// TIA Portal project "7_Height_Sorting_Basic" (V19)

(* hardware
DEVICE "S7-1500/ET200MP station_1"  S7-1500 station
   slot 0: "Rail_0"  Rack  6ES7 590-1***0-0AA0
   slot 1: "PLC_1"  CPU 1513-1 PN  6ES7 513-1AL02-0AB0  V2.9
      slot 3: "CPU display_1"  6ES7591-1AA00-0AA0
      slot 32768: "PROFINET interface_1"  X1
         slot 32769: "Port_1"  X1 P1
         slot 32770: "Port_2"  X1 P2
      slot 34817: "Virtual CP interface port_1"  Virtual CP interface port  Virtual CP interface port
*)

// ===== PLC "PLC_1"  CPU 1513-1 PN =====

VAR_GLOBAL   // PLC tag table "Default tag table"
   "Tag_1" AT %M0.0 : Bool;
   "Tag_2" AT %M0.1 : Bool;
   "Tag_3" AT %M0.2 : Bool;
   "Tag_4" AT %M0.3 : Bool;
   "Tag_5" AT %M0.4 : Bool;
   "Tag_6" AT %M0.5 : Bool;
   "Tag_7" AT %M2.1 : Bool;
   "Tag_8" AT %M1.7 : Bool;
   "Tag_9" AT %M2.0 : Bool;
   "Tag_10" AT %MW100 : Int;
   "Tag_11" AT %M2.2 : Bool;
   "Tag_12" AT %M1.0 : Bool;
   "Tag_13" AT %M1.1 : Bool;
   "Tag_14" AT %M1.4 : Bool;
   "Tag_15" AT %M1.2 : Bool;
   "Tag_16" AT %M1.3 : Bool;
   "Tag_17" AT %M1.5 : Bool;
   "Tag_18" AT %M1.6 : Bool;
   "Tag_19" AT %M2.4 : Bool;
   "Tag_20" AT %M2.5 : Bool;
END_VAR

VAR_GLOBAL   // PLC tag table "Tag table from XML_1"
   "Start Button" AT %I0.0 : Bool;
   "Stop Button" AT %I0.1 : Bool;
   "High Sensor" AT %I0.2 : Bool;
   "Low Sensor" AT %I0.3 : Bool;
   "Pallet sensor" AT %I0.4 : Bool;
   "Loaded" AT %I0.5 : Bool;
   "At right entry" AT %I0.6 : Bool;
   "At left entry" AT %I0.7 : Bool;
   "At right exit" AT %I1.0 : Bool;
   "At left exit" AT %I1.1 : Bool;
   "Start Button (LED)" AT %Q0.0 : Bool;
   "Stop Button (LED)" AT %Q0.1 : Bool;
   "Conveyor entry" AT %Q0.2 : Bool;
   "Conveyor right" AT %Q0.3 : Bool;
   "Conveyor left" AT %Q0.4 : Bool;
   "Load" AT %Q0.5 : Bool;
   "Transf. left" AT %Q0.6 : Bool;
   "Transf. right" AT %Q0.7 : Bool;
   "Right count" AT %QW30 : Int;
   "Left Count" AT %QW32 : Int;
END_VAR

// folder: System blocks/Program resources

DATA_BLOCK "IEC_Timer_0_DB"   // DB1
{ S7_Optimized_Access := 'TRUE' }
AUTHOR : Simatic
FAMILY : IEC
NAME : IEC_TMR
VERSION : 1.0
// stored: InstanceOfName IEC_TIMER
"IEC_TIMER"
BEGIN
END_DATA_BLOCK

DATA_BLOCK "IEC_Counter_0_DB"   // DB2
{ S7_Optimized_Access := 'TRUE' }
AUTHOR : Simatic
FAMILY : IEC
NAME : CNTR
VERSION : 1.0
// stored: InstanceOfName IEC_COUNTER
"IEC_COUNTER"
BEGIN
END_DATA_BLOCK

DATA_BLOCK "IEC_Counter_0_DB_1"   // DB3
{ S7_Optimized_Access := 'TRUE' }
AUTHOR : Simatic
FAMILY : IEC
NAME : CNTR
VERSION : 1.0
// stored: InstanceOfName IEC_COUNTER
"IEC_COUNTER"
BEGIN
END_DATA_BLOCK

DATA_BLOCK "IEC_Counter_0_DB_2"   // DB4
{ S7_Optimized_Access := 'TRUE' }
AUTHOR : Simatic
FAMILY : IEC
NAME : CNTR
VERSION : 1.0
// stored: InstanceOfName IEC_COUNTER
"IEC_COUNTER"
BEGIN
END_DATA_BLOCK

DATA_BLOCK "IEC_Counter_0_DB_3"   // DB5
{ S7_Optimized_Access := 'TRUE' }
AUTHOR : Simatic
FAMILY : IEC
NAME : CNTR
VERSION : 1.0
// stored: InstanceOfName IEC_COUNTER
"IEC_COUNTER"
BEGIN
END_DATA_BLOCK

// folder: (top level)

ORGANIZATION_BLOCK "Main"   // OB1, LAD, ProgramCycle
TITLE = "Main Program Sweep (Cycle)"
{ S7_Optimized_Access := 'TRUE' }
VERSION : 0.1
   VAR_INPUT
      Initial_Call : Bool;   // Initial call of this OB
      Remanence : Bool;   // =True, if remanent data are available
   END_VAR
   VAR_TEMP   // added for the SCL form of the ladder/FBD networks
      _w1 : Bool;
      _w2 : Bool;
      _w3 : Bool;
      _w4 : Bool;
   END_VAR
BEGIN

REGION Network 1: ON/OFF the LEDs
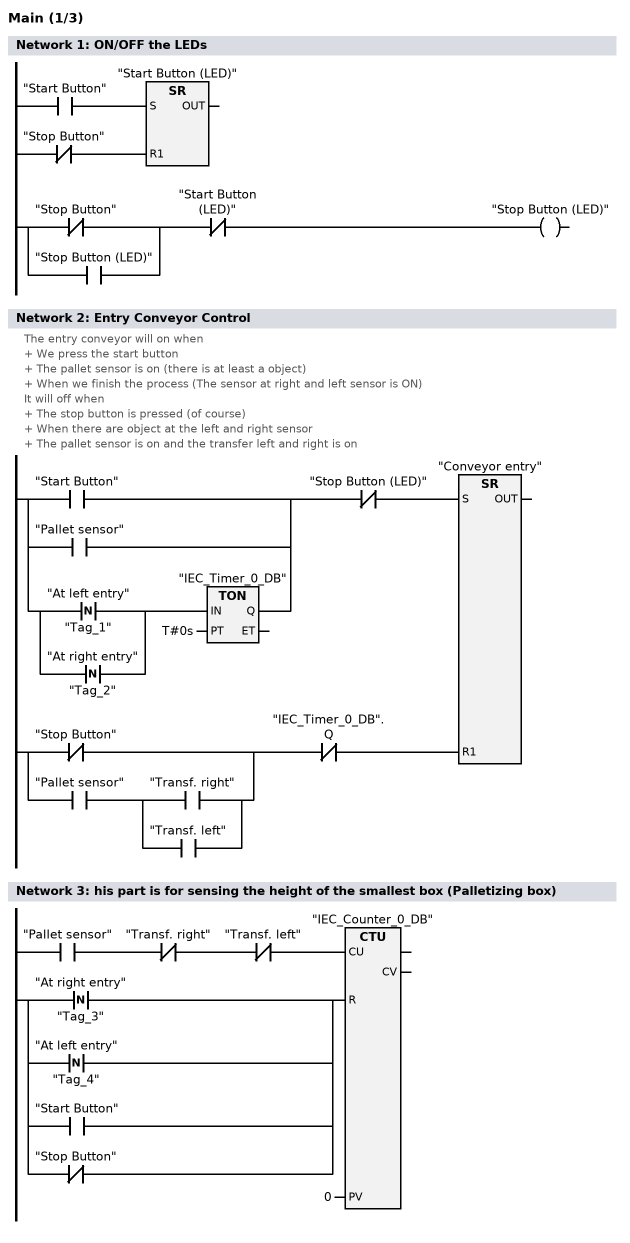
   RUNG wire#powerrail
      Contact( "Start Button" )
      S_SR(operand := "Start Button (LED)", r1 := wire#w1)
   END_RUNG
   RUNG wire#powerrail
      I_Contact( "Stop Button" )
   END_RUNG wire#w1
   RUNG wire#powerrail
      I_Contact( "Stop Button" )
      wire#w2
      I_Contact( "Start Button (LED)" )
      Coil( "Stop Button (LED)" )
   END_RUNG
   RUNG wire#powerrail
      Contact( "Stop Button (LED)" )
   END_RUNG wire#w2
   // the same network as SCL:
   IF "Start Button" THEN
       "Start Button (LED)" := TRUE;   // SR flip-flop
   END_IF;
   IF NOT "Stop Button" THEN "Start Button (LED)" := FALSE; END_IF;
   "Stop Button (LED)" := (NOT "Stop Button" OR "Stop Button (LED)") AND NOT "Start Button (LED)";
END_REGION

REGION Network 2: Entry Conveyor Control
   // The entry conveyor will on when
   // + We press the start button
   // + The pallet sensor is on (there is at least a object)
   // + When we finish the process (The sensor at right and left sensor is ON)
   // It will off when
   // + The stop button is pressed (of course)
   // + When there are object at the left and right sensor
   // + The pallet sensor is on and the transfer left and right is on
   #_w1 := NOT "At left entry" AND "Tag_1";   // falling edge of "At left entry"
   "Tag_1" := "At left entry";
   #_w2 := NOT "At right entry" AND "Tag_2";   // falling edge of "At right entry"
   "Tag_2" := "At right entry";
   "IEC_Timer_0_DB".TON(IN := #_w1 OR #_w2, PT := T#0s);
   IF ("Start Button" OR "Pallet sensor" OR "IEC_Timer_0_DB".Q) AND NOT "Stop Button (LED)" THEN
       "Conveyor entry" := TRUE;   // SR flip-flop
   END_IF;
   IF (NOT "Stop Button" OR ("Pallet sensor" AND ("Transf. right" OR "Transf. left"))) AND NOT "IEC_Timer_0_DB".Q THEN
       "Conveyor entry" := FALSE;
   END_IF;
END_REGION

REGION Network 3: his part is for sensing the height of the smallest box (Palletizing box)
   #_w1 := NOT "At right entry" AND "Tag_3";   // falling edge of "At right entry"
   "Tag_3" := "At right entry";
   #_w2 := NOT "At left entry" AND "Tag_4";   // falling edge of "At left entry"
   "Tag_4" := "At left entry";
   "IEC_Counter_0_DB".CTU(CU := "Pallet sensor" AND NOT "Transf. right" AND NOT "Transf. left",
                          R := #_w1 OR #_w2 OR "Start Button" OR NOT "Stop Button",
                          PV := 0);
END_REGION

REGION Network 4: This part for box size S and M
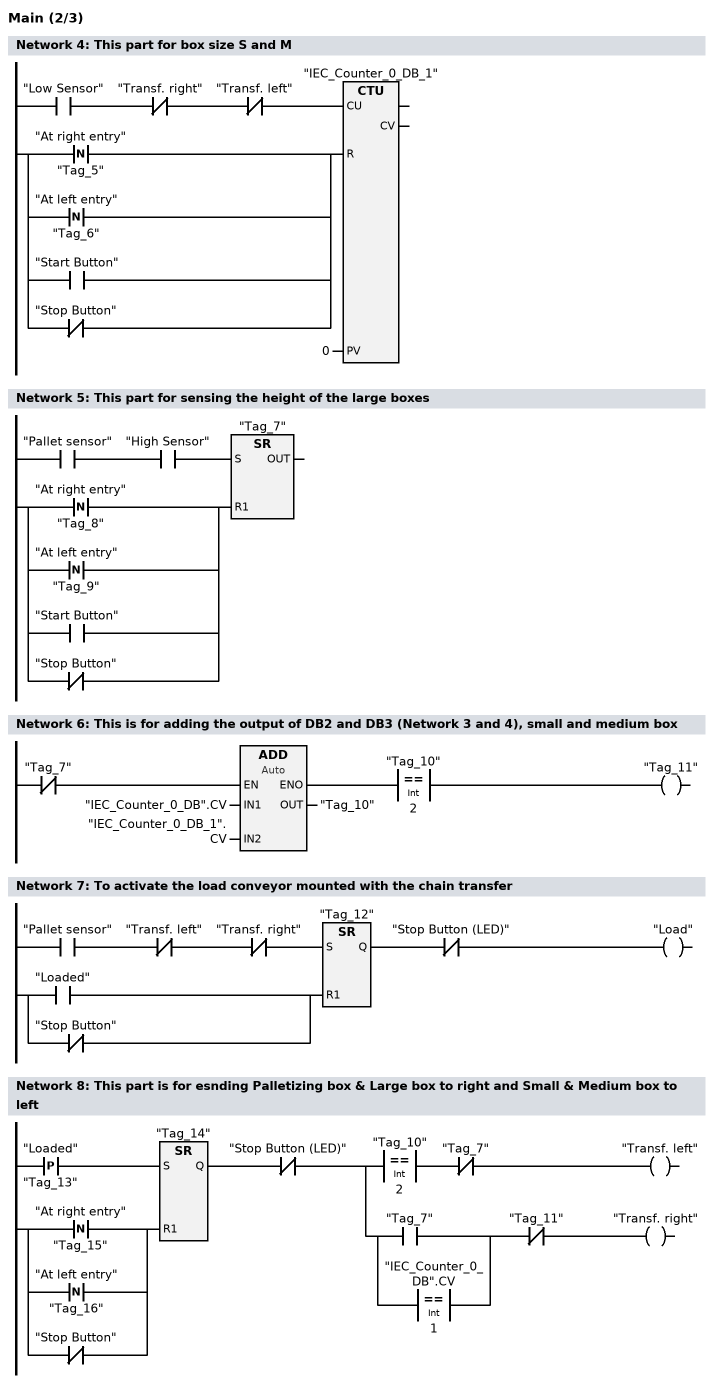
   #_w1 := NOT "At right entry" AND "Tag_5";   // falling edge of "At right entry"
   "Tag_5" := "At right entry";
   #_w2 := NOT "At left entry" AND "Tag_6";   // falling edge of "At left entry"
   "Tag_6" := "At left entry";
   "IEC_Counter_0_DB_1".CTU(CU := "Low Sensor" AND NOT "Transf. right" AND NOT "Transf. left",
                           R := #_w1 OR #_w2 OR "Start Button" OR NOT "Stop Button",
                           PV := 0);
END_REGION

REGION Network 5: This part for sensing the height of the large boxes
   RUNG wire#powerrail
      Contact( "Pallet sensor" )
      Contact( "High Sensor" )
      S_SR(operand := "Tag_7", r1 := wire#w1)
   END_RUNG
   RUNG wire#powerrail
      N_Contact(operand := "At right entry", bit := "Tag_8")
   END_RUNG wire#w1
   RUNG wire#powerrail
      N_Contact(operand := "At left entry", bit := "Tag_9")
   END_RUNG wire#w1
   RUNG wire#powerrail
      Contact( "Start Button" )
   END_RUNG wire#w1
   RUNG wire#powerrail
      I_Contact( "Stop Button" )
   END_RUNG wire#w1
   // the same network as SCL:
   #_w1 := NOT "At right entry" AND "Tag_8";   // falling edge of "At right entry"
   "Tag_8" := "At right entry";
   #_w2 := NOT "At left entry" AND "Tag_9";   // falling edge of "At left entry"
   "Tag_9" := "At left entry";
   IF "Pallet sensor" AND "High Sensor" THEN
       "Tag_7" := TRUE;   // SR flip-flop
   END_IF;
   IF #_w1 OR #_w2 OR "Start Button" OR NOT "Stop Button" THEN "Tag_7" := FALSE; END_IF;
END_REGION

REGION Network 6: This is for adding the output of DB2 and DB3 (Network 3 and 4), small and medium box
   RUNG wire#powerrail
      I_Contact( "Tag_7" )
      Add(in1 := "IEC_Counter_0_DB".CV, in2 := "IEC_Counter_0_DB_1".CV, out => "Tag_10")
      { S7_Templates := "SrcType := Int" } EQ_Contact(in1 := "Tag_10", in2 := 2)
      Coil( "Tag_11" )
   END_RUNG
   // the same network as SCL:
   IF NOT "Tag_7" THEN "Tag_10" := "IEC_Counter_0_DB".CV + "IEC_Counter_0_DB_1".CV; END_IF;
   "Tag_11" := NOT "Tag_7" AND ("Tag_10" = 2);
END_REGION

REGION Network 7: To activate the load conveyor mounted with the chain transfer
   RUNG wire#powerrail
      Contact( "Pallet sensor" )
      I_Contact( "Transf. left" )
      I_Contact( "Transf. right" )
      S_SR(operand := "Tag_12", r1 := wire#w1)
      I_Contact( "Stop Button (LED)" )
      Coil( "Load" )
   END_RUNG
   RUNG wire#powerrail
      Contact( "Loaded" )
   END_RUNG wire#w1
   RUNG wire#powerrail
      I_Contact( "Stop Button" )
   END_RUNG wire#w1
   // the same network as SCL:
   IF "Pallet sensor" AND NOT "Transf. left" AND NOT "Transf. right" THEN
       "Tag_12" := TRUE;   // SR flip-flop
   END_IF;
   IF "Loaded" OR NOT "Stop Button" THEN "Tag_12" := FALSE; END_IF;
   "Load" := "Tag_12" AND NOT "Stop Button (LED)";
END_REGION

REGION Network 8: This part is for esnding Palletizing box & Large box to right and Small & Medium box to left
   RUNG wire#powerrail
      P_Contact(operand := "Loaded", bit := "Tag_13")
      S_SR(operand := "Tag_14", r1 := wire#w1)
      I_Contact( "Stop Button (LED)" )
      wire#w2
      { S7_Templates := "SrcType := Int" } EQ_Contact(in1 := "Tag_10", in2 := 2)
      I_Contact( "Tag_7" )
      Coil( "Transf. left" )
   END_RUNG
   RUNG wire#powerrail
      N_Contact(operand := "At right entry", bit := "Tag_15")
   END_RUNG wire#w1
   RUNG wire#powerrail
      N_Contact(operand := "At left entry", bit := "Tag_16")
   END_RUNG wire#w1
   RUNG wire#powerrail
      I_Contact( "Stop Button" )
   END_RUNG wire#w1
   RUNG wire#w2
      Contact( "Tag_7" )
      wire#w3
      I_Contact( "Tag_11" )
      Coil( "Transf. right" )
   END_RUNG
   RUNG wire#w2
      { S7_Templates := "SrcType := Int" } EQ_Contact(in1 := "IEC_Counter_0_DB".CV, in2 := 1)
   END_RUNG wire#w3
   // the same network as SCL:
   #_w1 := "Loaded" AND NOT "Tag_13";   // rising edge of "Loaded"
   "Tag_13" := "Loaded";
   #_w2 := NOT "At right entry" AND "Tag_15";   // falling edge of "At right entry"
   "Tag_15" := "At right entry";
   #_w3 := NOT "At left entry" AND "Tag_16";   // falling edge of "At left entry"
   "Tag_16" := "At left entry";
   IF #_w1 THEN
       "Tag_14" := TRUE;   // SR flip-flop
   END_IF;
   IF #_w2 OR #_w3 OR NOT "Stop Button" THEN "Tag_14" := FALSE; END_IF;
   #_w4 := "Tag_14" AND NOT "Stop Button (LED)";
   "Transf. left" := #_w4 AND ("Tag_10" = 2) AND NOT "Tag_7";
   "Transf. right" := #_w4 AND ("Tag_7" OR ("IEC_Counter_0_DB".CV = 1)) AND NOT "Tag_11";
END_REGION

REGION Network 9: To activate or deactivate the conveyor right (CR)
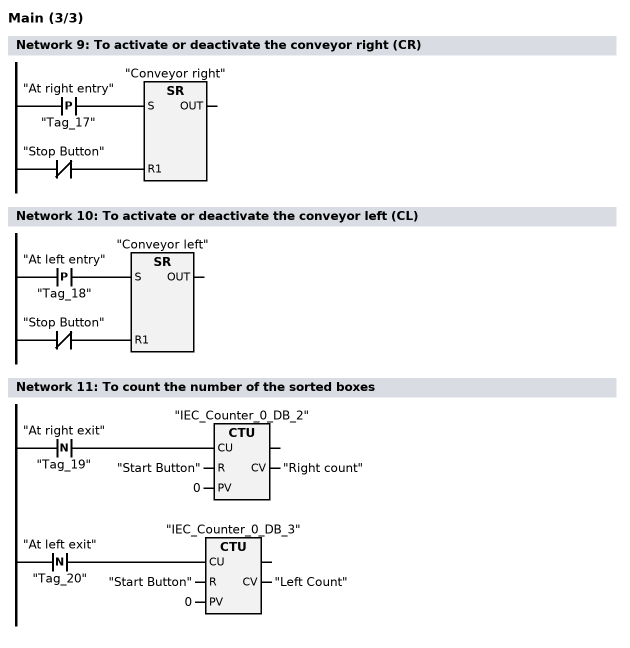
   RUNG wire#powerrail
      P_Contact(operand := "At right entry", bit := "Tag_17")
      S_SR(operand := "Conveyor right", r1 := wire#w1)
   END_RUNG
   RUNG wire#powerrail
      I_Contact( "Stop Button" )
   END_RUNG wire#w1
   // the same network as SCL:
   #_w1 := "At right entry" AND NOT "Tag_17";   // rising edge of "At right entry"
   "Tag_17" := "At right entry";
   IF #_w1 THEN
       "Conveyor right" := TRUE;   // SR flip-flop
   END_IF;
   IF NOT "Stop Button" THEN "Conveyor right" := FALSE; END_IF;
END_REGION

REGION Network 10: To activate or deactivate the conveyor left (CL)
   RUNG wire#powerrail
      P_Contact(operand := "At left entry", bit := "Tag_18")
      S_SR(operand := "Conveyor left", r1 := wire#w1)
   END_RUNG
   RUNG wire#powerrail
      I_Contact( "Stop Button" )
   END_RUNG wire#w1
   // the same network as SCL:
   #_w1 := "At left entry" AND NOT "Tag_18";   // rising edge of "At left entry"
   "Tag_18" := "At left entry";
   IF #_w1 THEN
       "Conveyor left" := TRUE;   // SR flip-flop
   END_IF;
   IF NOT "Stop Button" THEN "Conveyor left" := FALSE; END_IF;
END_REGION

REGION Network 11: To count the number of the sorted boxes
   #_w1 := NOT "At right exit" AND "Tag_19";   // falling edge of "At right exit"
   "Tag_19" := "At right exit";
   "IEC_Counter_0_DB_2".CTU(CU := #_w1, R := "Start Button", PV := 0, CV => "Right count");
   #_w2 := NOT "At left exit" AND "Tag_20";   // falling edge of "At left exit"
   "Tag_20" := "At left exit";
   "IEC_Counter_0_DB_3".CTU(CU := #_w2, R := "Start Button", PV := 0, CV => "Left Count");
END_REGION
END_ORGANIZATION_BLOCK